// TIA Portal V17 export
// export: Created 2025-05-22T06:01:47.7948511Z, ExportSetting WithDefaults, DisplayName Totally Integrated Automation Portal, DisplayVersion V17 Update 8, DisplayName TIA Portal Openness, DisplayVersion V17 Update 8, DisplayName TIA Portal Version Control Interface, DisplayVersion V17, DisplayName SINAMICS Startdrive Advanced, DisplayVersion V17 SP2, DisplayName SINAMICS Startdrive G110M, G120, G120C, G120D, G120P, G115D, DisplayVersion V17 SP2, DisplayName SINAMICS Startdrive G130, G150, S120, S150, SINAMICS MV, S210, DisplayVersion V17 SP2, DisplayName STEP 7 Professional, DisplayVersion V17 Update 8, DisplayName SINUMERIK ONE STEP 7 Toolbox, DisplayVersion V17 Update 12, DisplayName SINUMERIK ONE PLC Basic Program Plus, DisplayVersion V17 Update 12, DisplayName SINUMERIK 840D sl STEP 7 Toolbox, DisplayVersion V17 Update 12, DisplayName STEP 7 Safety, DisplayVersion V17 Update 6, DisplayName WinCC Advanced, DisplayVersion V17 Update 8
TYPE "FIXTURE_STATUS"
// stored: IsFailsafeCompliant false
   STRUCT
      INPUT_PART_A_PRESENT : Bool;   // FIXTURE INPUT PART A PRESENT
      INPUT_PART_A_PRESENT_FACE_TYPE : Bool;   // FIXTURE INPUT PART A PRESENT FIXTURE FACE TYPE UP
      INPUT_PART_A_PRESENT_MEM : Bool;   // FIXTURE INPUT PART A PRESENT MEMORY
      INPUT_PART_A_PRESENT_FACE_TYPE_MEM : Bool;   // FIXTURE INPUT PART A PRESENT FIXTURE FACE TYPE UP MEMORY
      CLAMPED_WITH_PART_A : Bool;   // FIXTURE CLAMPED WITH PART A
      CLAMPED_WITHOUT_PART_A : Bool;   // FIXTURE CLAMPED WITHOUT PART A
      CLAMPED_WITH_PARTS : Bool;   // FIXTURE CLAMPED WITH PARTS
      CLAMPED_WITHOUT_PARTS : Bool;   // FIXTURE CLAMPED WITHOUT PARTS
      PARTIAL_CLAMPED : Bool;   // FIXTURE PARTIAL CLAMPED
      CLAMPED_WITH_PART_ANALOG : Bool;   // FIXTURE CLAMPED WITH PART ANALOG
      CLAMPED_OK : Bool;   // FIXTURE CLAMPED OK
      CLAMPED_DELAYED : Bool;   // FIXTURE CLAMPED DELAYED
      CLAMPED_WITHOUT_PART_ANALOG : Bool;   // FIXTURE CLAMPED WITHOUT PART ANALOG
      UNCLAMPED_ANALOG : Bool;   // FIXTURE UNCLAMPED
      FIXTURE_NOT_CLAMPED_ALARM : Bool;   // FIXTURE NOT CLAMPED DURING MACHINING ALARM
      PART_A_PRESENT_DISCORDANCY : Bool;   // FIXTURE PART A PRESENT DISCORDANCY
      PART_A_ORIENTATED_DISCORDANCY : Bool;   // FIXTURE PART A ORIENTATED DISCORDANCY
      PART_TYPE_DISCORDANCY : Bool;   // FIXTURE PART TYPE DISCORDANCY
      ANY_PART_PRESENT : Bool;   // FIXTURE ANY PART PRESENT
      CLAMPED_MEMORY_DONE : Bool;   // FIXTURE CLAMPED MEMORY DONE
      AUX_1 : Bool;
      AUX_2 : Bool;
      AUX_3 : Bool;
      TIMER_CLAMPED_DELAY : TON_TIME;   // FIXTURE CLAMPED TIMER
      TIMER_PART_A_ORIENTATION { S7_SetPoint := 'True'} : TON_TIME;   // FIXTURE PART A ORIENTATION TIMER
      TIMER_PART_A_DISCORDANCY { S7_SetPoint := 'True'} : TON_TIME;   // FIXTURE PART A DISCORDANCY TIMER
      TIMER_CLAMPED_WITH_ANALOG { S7_SetPoint := 'True'} : TOF_TIME;
   END_STRUCT;
   // TIMER_PART_A_ORIENTATION.PT := T#750ms;
   // TIMER_PART_A_DISCORDANCY.PT := T#750ms;
   // TIMER_CLAMPED_WITH_ANALOG.PT := T#100ms;
END_TYPE
